{attribute 'no_explicit_call' := 'Do not call the body - Stick to OOP'}
FUNCTION_BLOCK FB_GigeCamera_Any EXTENDS FB_CH_Object IMPLEMENTS I_GevCameraControl, I_GigE_Beckhoff_Standalone, I_GetImage
VAR
	// This FB provides the basic functionality to control a GigE Vision camera and access its calibration data.
	fbCamera 						: FB_VN_GevCameraControl;	
	fbTriggerEtherCat				: FB_EtherCAT_Timestamp;
	
	{attribute 'hide'}	
	bInSimulation 					: BOOL;
	{attribute 'hide'}	
	eCameraType						: E_CameraType; 	
	{attribute 'hide'}
	fbGigeAnyRegister			 			: FB_GigE_Register_Any(ipCamera := THIS^);
	{attribute 'hide'}
	fbGigeBeckhoffRegisterVCS2xxx 			: FB_GigE_Register_Beckhoff_VCS2xxx(ipCamera := THIS^);
	{attribute 'hide'}
	fbGigeBeckhoffRegisterVUI2xxx 			: FB_GigE_Register_Beckhoff_VUI2xxx(ipCamera := THIS^);
	{attribute 'hide'}	
	ipRegister 								: I_GigeRegisterBase := fbGigeAnyRegister;
		
	{attribute 'hide'}	
	bInitDone 			: BOOL;
	{attribute 'hide'}
	bResetCommand		: BOOL;
	{attribute 'hide'}  						
	fbFeedback 			: FB_CH_Feedback(THIS^.fbSourceInfo); 
	{attribute 'hide'}
	fbAlarmOidNotSet 	: FB_TcAlarm;									// Alarm due to source state
	{attribute 'hide'}
	fbEthernetLinkDown 	: FB_TcAlarm;									// Camera is not connectode or has no power
	
	//TcCom object Camera
	{attribute 'hide'}
	ipGevImageProviderComObject 		: ITComObject;	
	{attribute 'hide'}
	ipGevImageAcquisitionComObject 		: ITComObject;	
	{attribute 'hide'}
	ipIpStackComObject 					: ITComObject;			
END_VAR

{attribute 'monitoring' := 'call'}
//Once as a Beckhoff camera is detected at startup, the corresponding type is loaded automatically. 
PROPERTY CameraType : E_CameraType
GET
CameraType := THIS^.eCameraType;
END_GET
SET
//if a new type is selectet, init the last one to reset all errors
IF (THIS^.CameraType <> THIS^.eCameraType) AND (THIS^.ipRegister <> 0) THEN
	THIS^.ipRegister.Initialize();
END_IF

//store new type
THIS^.eCameraType := CameraType;

//write new object to interface
CASE THIS^.eCameraType OF	
	E_CameraType.Beckhoff_VCS2xxx:
		THIS^.ipRegister := THIS^.fbGigeBeckhoffRegisterVCS2xxx;
		
	E_CameraType.Beckhoff_VUI2xxx:
		THIS^.ipRegister := THIS^.fbGigeBeckhoffRegisterVUI2xxx;
	
	ELSE
		THIS^.ipRegister := THIS^.fbGigeAnyRegister;;
END_CASE
END_SET
END_PROPERTY

//	The connection to the camera has been established. Gige-Vision parameters can now be read or written
{attribute 'monitoring' := 'call'}
PROPERTY ControlChannelOpen : BOOL
GET
CASE THIS^.State OF
	TCVN_CS_ERROR, TCVN_CS_INITIAL, TCVN_CS_INITIALIZING, TCVN_CS_INITIALIZED,TCVN_CS_OPENING,TCVN_CS_CLOSING:
		ControlChannelOpen := FALSE;
	
	TCVN_CS_OPENED, TCVN_CS_STARTACQUISITION,  TCVN_CS_ACQUIRING, TCVN_CS_STOPACQUISITION, TCVN_CS_RESETTINGFEATURES, TCVN_CS_TRIGGERING:
		ControlChannelOpen := TRUE;

	ELSE
		;//Unknown
END_CASE
END_GET
END_PROPERTY

METHOD FB_exit : BOOL
VAR_INPUT
	bInCopyCode : BOOL; // if TRUE, the exit method is called for exiting an instance that is copied afterwards (online change).
END_VAR
//Not on onlinechange
IF NOT bInCopyCode THEN
	IF THIS^.ipGevImageProviderComObject <> 0 THEN
		FW_SafeRelease(ADR(ipGevImageProviderComObject));
		FW_SafeRelease(ADR(ipGevImageAcquisitionComObject));
		FW_SafeRelease(ADR(ipIpStackComObject));
	END_IF	
END_IF
END_METHOD

METHOD FB_init : BOOL
VAR_INPUT
	bInitRetains : BOOL; // if TRUE, the retain variables are initialized (warm start / cold start)
	bInCopyCode : BOOL;  // if TRUE, the instance afterwards gets moved into the copy code (online change)
END_VAR
VAR
	fbGetCurTaskIdx  : GETCURTASKINDEX;
END_VAR
IF NOT bInCopyCode THEN
	//Start with an unknown camera. 
	//Once as a Beckhoff camera is detected, the corresponding type is loaded automatically. 
	THIS^.CameraType := E_CameraType.Unknown;
END_IF
END_METHOD

{attribute 'monitoring':='call'}
PROPERTY Feedback : I_CH_Feedback
GET
Feedback := THIS^.fbFeedback;
END_GET
END_PROPERTY

{attribute 'monitoring' := 'call'}
// This FB provides the basic functionality to control a GigE Vision camera and access its calibration data.
PROPERTY GevCameraControl : REFERENCE TO FB_VN_GevCameraControl
GET
GevCameraControl REF= THIS^.fbCamera;
END_GET
END_PROPERTY

METHOD Initialize : HRESULT
VAR 
	fbTaskInfo			: PlcTaskSystemInfo;
	nOid : OTCID;	
	nParaSize : UDINT;
	pParaData : PVOID;
	hr : HRESULT;
END_VAR
VAR_INST
	//This error cannot be reset. Requires a reset cold
	{attribute 'hide'}	
	fbInitError : FB_TcAlarm;
END_VAR
VAR CONSTANT
	N_IDX_OFFSET_GevImageAcquisition 	: UDINT := 16#00000001;
	N_IDX_OFFSET_IP_STACK 				: UDINT := 16#00000013;
END_VAR
hr := SUPER^.Initialize();


// Object id of ImagePoovider is not set
IF THIS^.fbCamera.oidITcVnGevImageProvider = 0 THEN
	IF NOT fbInitError.bRaised THEN 
		//This error cannot be reset. Requires a reset cold
		fbInitError.CreateEx(stEventEntry:=TC_EVENTS.CHALET_Vision_Events.ObjectIdNotSet, ipSourceInfo := THIS^.fbSourceInfo, bWithConfirmation := FALSE);
		fbInitError.Raise(0);
	END_IF
	Initialize := E_FAIL;
	RETURN;
END_IF


//Read information from TcCom object
//Get interface to ComObject
hr := FW_ObjMgr_GetObjectInstance(oid:= THIS^.OID, iid:= TC_GLOBAL_IID_LIST.IID_ITComObject, pipUnk:= ADR(THIS^.ipGevImageProviderComObject));
IF THIS^.ipGevImageProviderComObject <> 0 THEN
	//Read object id of TcCom GevImageAcquisitionComObject
	nOid := 0;
	nParaSize := SIZEOF(nOid);	pParaData := ADR(nOid);
	hr := ipGevImageProviderComObject.TcGetObjPara(pid:=N_IDX_OFFSET_GevImageAcquisition , nData:= nParaSize, pData:= pParaData, pgp:=0 );
	
	//Get interface of GevImageAcquisition
	hr := FW_ObjMgr_GetObjectInstance(oid:= nOid, iid:= TC_GLOBAL_IID_LIST.IID_ITComObject, pipUnk:= ADR(THIS^.ipGevImageAcquisitionComObject));
	IF THIS^.ipGevImageAcquisitionComObject <> 0 THEN
		//Read object id of TcCom 
		nOid := 0;
		nParaSize := SIZEOF(nOid);	pParaData := ADR(nOid);
		hr := ipGevImageAcquisitionComObject.TcGetObjPara(pid:=N_IDX_OFFSET_IP_STACK , nData:= nParaSize, pData:= pParaData, pgp:=0 );
		// If IP-Stack was not found in GevImageAcquisitionComObject then camera is in simulation mode
		IF hr = S_OK THEN
			//get interface to ipstack
			hr := FW_ObjMgr_GetObjectInstance(oid:= nOid, iid:= TC_GLOBAL_IID_LIST.IID_ITComObject, pipUnk:= ADR(THIS^.ipIpStackComObject));
		ELSE
			bInSimulation := TRUE;
			hr := S_OK;
		END_IF
	END_IF
END_IF


//Subelement
hr := GetMostSignificant(hr, fbTriggerEtherCat.Initialize());
IF THIS^.ipRegister <> 0 THEN
	hr := GetMostSignificant(hr, THIS^.ipRegister.Initialize());
END_IF


Initialize := hr;

IF Initialize = S_OK THEN
	THIS^.bInitDone := TRUE;
END_IF
END_METHOD

{attribute 'monitoring':='call'}
PROPERTY Initialized : BOOL
GET
Initialized := THIS^.bInitDone;
END_GET
END_PROPERTY

{attribute 'monitoring' := 'call'}
//Returns the OTCID OF the camera object.
PROPERTY OID : CHALET_BaseComponents.OTCID
GET
OID := THIS^.fbCamera.oidITcVnGevImageProvider;
END_GET
END_PROPERTY

{attribute 'monitoring' := 'call'}
// Module started successfully and entered aquiring mode
PROPERTY PUBLIC Operational : BOOL
GET
VAR
	eState : ETcVnCameraState;
END_VAR
eState := THIS^.State;
Operational := (eState = TCVN_CS_ACQUIRING) OR (eState = TCVN_CS_TRIGGERING);
END_GET
END_PROPERTY

{attribute 'monitoring' := 'call'}
//Access to the important parameters marked as standard in Gige-Vision
PROPERTY RegisterAnyCamera : I_GigE_Any_Camera
GET
//Convert in requestet interface
__QUERYINTERFACE(THIS^.ipRegister, RegisterAnyCamera);
END_GET
END_PROPERTY

{attribute 'monitoring' := 'call'}
//Interface to the parameters, can be 0(=invalid interface) depending on the hardware
PROPERTY RegisterBeckhoffCamera : I_GigE_Beckhoff_Camera
GET
//Convert in requestet interface
__QUERYINTERFACE(THIS^.ipRegister, RegisterBeckhoffCamera);
END_GET
END_PROPERTY

{attribute 'monitoring' := 'call'}
//Interface to the parameters, can be 0(=invalid interface) depending on the hardware
PROPERTY RegisterLighting : I_GigE_Beckhoff_Lighting
GET
//Convert in requestet interface
__QUERYINTERFACE(THIS^.ipRegister, RegisterLighting);
END_GET
END_PROPERTY

{attribute 'monitoring' := 'call'}
//Interface to the parameters, can be 0(=invalid interface) depending on the hardware
PROPERTY RegisterOpticControl : I_GigE_Beckhoff_OpticControl
GET
//Convert in requestet interface
__QUERYINTERFACE(THIS^.ipRegister, RegisterOpticControl);
END_GET
END_PROPERTY

//Try to reset the camera connection
METHOD Reset : HRESULT
VAR_INPUT
END_VAR
THIS^.bResetCommand := TRUE;

fbFeedback.ActiveCommand := 'Reset';
fbFeedback.LastCommandAccepted	:= TRUE;
fbFeedback.hr := THIS^.fbCamera.Reset();
END_METHOD

{attribute 'monitoring' := 'call'}
//Simulation mode is active
PROPERTY Simulation : BOOL
GET
Simulation := bInSimulation;
END_GET
END_PROPERTY

{attribute 'monitoring' := 'call'}
//Gets the current state of the internal camera control state machine.
PROPERTY State : ETcVnCameraState
GET
State := THIS^.fbCamera.GetState();
END_GET
END_PROPERTY

{attribute 'monitoring' := 'call'}
//Access to the interface to control the EtherCAT timestamp trigger
PROPERTY TriggerEtherCat : I_EtherCat_Trigger
GET
TriggerEtherCat := THIS^.fbTriggerEtherCat;
END_GET
END_PROPERTY

//Send the 'SoftwareTriggerCommands' defined in the TcVnGevImageProvider TcCOM module to the camera.
METHOD PUBLIC TriggerSoftware : HRESULT
VAR
	eState : ETcVnCameraState;
END_VAR
eState := THIS^.State;

(* Check if not in wrong state *)
IF NOT ((eState = ETcVnCameraState.TCVN_CS_ACQUIRING) OR (eState = ETcVnCameraState.TCVN_CS_OPENED) OR THIS^.Simulation) THEN
	TriggerSoftware := E_FAIL;
	RETURN;
END_IF

// Trigger image
fbFeedback.ActiveCommand := 'TriggerImage';
fbFeedback.LastCommandAccepted	:= TRUE;
fbFeedback.hr := fbCamera.TriggerImage();
TriggerSoftware := fbFeedback.hr;
END_METHOD

//Gets the current available image (first in receive queue) and its corresponding GVSP info
METHOD TryGetImage : HRESULT
VAR_INPUT
	stImageWithInfo : REFERENCE TO ST_ImageWithInfo;
END_VAR
VAR_INST
	{attribute 'hide'}							
    fbCrititcalSection : FB_IecCriticalSection;    						// Internal lock for test & set function    
END_VAR
VAR
	ipImageTemp   : ITcVnImage;
	stGvspInfoTemp : GVSP_IMAGE_INFO;
END_VAR
IF NOT __ISVALIDREF(stImageWithInfo) THEN
	//Error, invalide input
	TryGetImage := E_FAIL;
	RETURN;
END_IF


(*  Lock the image to prevent multiple access *)
(*	🔒 LOCKED FROM HERE --------------------------------------------- *)
IF fbCrititcalSection.Enter() THEN
	
	(* Get current image from camera and store result in temp variable*)
	TryGetImage := fbCamera.GetCurrentImageWithGvspInfo(
						ipImage := ipImageTemp,
						stGvspInfo := stGvspInfoTemp
						);
					
	(* If new image found *)				
	IF TryGetImage = S_OK THEN
		
		(* Release the old image before overwriting it with the new one *)	
		IF stImageWithInfo.ipImage <> 0 THEN
			FW_SafeRelease(ADR(stImageWithInfo.ipImage));
		END_IF		
	
		//Handover new data
		stImageWithInfo.ipImage 		:= ipImageTemp;
		stImageWithInfo.stGvspInfo 		:= stGvspInfoTemp;

		(*For a camera a fictitious name *)
		stImageWithInfo.sCurrentImageFileName := TO_STRING(stImageWithInfo.stGvspInfo.BlockId);		

		
		(* Get image info from received image *)
		F_VN_GetImageInfo(	ipImage:=stImageWithInfo.ipImage, 
							stImageInfo:=stImageWithInfo.stInfo, 
							hrPrev:=TryGetImage );	
	END_IF



	(*	🔓 LOCKED TO HERE ----------------------------------------------- *)
	fbCrititcalSection.Leave();
END_IF
END_METHOD

METHOD Update : HRESULT
VAR
	ipVnRegisterStatus : I_VnRegister;
	bAllReadDone : BOOL := TRUE;
	bAllWriteDone : BOOL := TRUE;
	nParaSize : UDINT;
	pParaData : PVOID;
	hr : HRESULT;
	stIpStackData : ST_IpStackDiag;
	bLinkDetected : BOOL;
	bParaReadSuccessful : BOOL;
END_VAR
VAR CONSTANT
	N_IDX_OFFSET_IP_STACK 	: UDINT := 16#03011108; // Parameter(online) in Planar Track object
END_VAR
//Force to initialize first
IF NOT THIS^.Initialized THEN
	THIS^.Initialize();
	RETURN;
END_IF


(* Source state machine *)
CASE THIS^.State OF
	TCVN_CS_INITIAL, TCVN_CS_INITIALIZING:
		fbFeedback.ActiveCommand := 'InitializeCamera';
		fbFeedback.hr := fbCamera.InitializeCamera();

	TCVN_CS_INITIALIZED,  TCVN_CS_OPENING:	
		IF THIS^.ipRegister <> 0 THEN
			//Redo a read or write for each parameter
			THIS^.ipRegister.RewriteParameters();
		END_IF
		fbFeedback.ActiveCommand := 'OpenCamera';
		fbFeedback.hr := fbCamera.OpenCamera();
		
	TCVN_CS_OPENED:
		(* Detect camera model once if unknown *)
		IF THIS^.CameraType = E_CameraType.Unknown AND THIS^.RegisterAnyCamera <> 0 AND THIS^.ipRegister.AllReadDone THEN
			IF FIND(THIS^.RegisterAnyCamera.DeviceModeNamel, 'VCS2') <> 0 THEN
				THIS^.CameraType := E_CameraType.Beckhoff_VCS2xxx;
			ELSIF FIND(THIS^.RegisterAnyCamera.DeviceModeNamel, 'VUI2') <> 0 THEN
				THIS^.CameraType := E_CameraType.Beckhoff_VUI2xxx;
			ELSE
				THIS^.CameraType := E_CameraType.ThirdParty;
			END_IF
		END_IF
		
		IF THIS^.Simulation THEN
			; //Stay in this state in Simulationmode	
		
		ELSIF THIS^.ipRegister = 0 THEN
			fbFeedback.ActiveCommand := 'StartAcquisition';
			fbFeedback.hr := fbCamera.StartAcquisition();
			
		ELSIF THIS^.ipRegister.AllReadDone AND THIS^.ipRegister.AllWriteDone THEN
			fbFeedback.ActiveCommand := 'StartAcquisition';
			fbFeedback.hr := fbCamera.StartAcquisition();

		ELSE	
			//Read and write all camera parameter in this OPENED-State 
			fbFeedback.ActiveCommand := 'ReadWrite camera parameters';
			fbFeedback.Busy	:= TRUE;
		END_IF
	
		
	TCVN_CS_STARTACQUISITION:
		fbFeedback.ActiveCommand := 'StartAcquisition';
		fbFeedback.hr := fbCamera.StartAcquisition();
		
		
	TCVN_CS_STOPACQUISITION:
		fbFeedback.ActiveCommand := 'StopAcquisition';
		fbFeedback.hr := fbCamera.StopAcquisition();
		
	TCVN_CS_ACQUIRING:
		;//wait for trigger
		
		//Check if a chage in opened state is required to read/write parameter
		IF VisionParameterlist.B_LEAVE_AQUIRRING_STATE_TO_WRITE_PARAMETER AND THIS^.ipRegister <> 0 AND_THEN NOT THIS^.ipRegister.AllWriteDone THEN
			fbFeedback.ActiveCommand := 'StopAcquisition';
			fbCamera.StopAcquisition();
		END_IF
		
	TCVN_CS_TRIGGERING:
		(* Execute the triggering until done *)
		fbFeedback.ActiveCommand := 'TriggerImage';
		fbFeedback.hr := fbCamera.TriggerImage();
		
	TCVN_CS_ERROR:	
		(* Reset if commanded *)
		IF THIS^.bResetCommand THEN
			fbFeedback.ActiveCommand := 'Reset';
			fbFeedback.hr := THIS^.fbCamera.Reset();			
		END_IF
		
END_CASE

(* Clear reset request if not in Error-State *)
IF THIS^.State <> TCVN_CS_ERROR THEN
	THIS^.bResetCommand := FALSE;
END_IF




// --- Write diagnostic information to eventloger
IF THIS^.State = TCVN_CS_ERROR AND VisionParameterlist.B_ALARM_IF_LINK_TO_CAMERA_IS_DOWN THEN
	//check IP-Stack an check if camera is conected	
	IF THIS^.ipIpStackComObject <> 0 THEN
		//Read object id of ipStack TcCom 
		nParaSize := SIZEOF(stIpStackData);	pParaData := ADR(stIpStackData);
		hr := ipIpStackComObject.TcGetObjPara(	pid		:=N_IDX_OFFSET_IP_STACK , 
												nData	:= nParaSize, 
												pData	:= pParaData, 
												pgp		:=0 );
		
		 // Link is active on uneven cts of linkchanges
		bLinkDetected := (stIpStackData.nLinkStatusChangedCnt MOD 2) = 1;
		bParaReadSuccessful := hr = S_OK;
		IF NOT THIS^.Simulation AND bParaReadSuccessful AND NOT bLinkDetected AND NOT fbEthernetLinkDown.bRaised THEN
			fbEthernetLinkDown.CreateEx(stEventEntry 		:= TC_EVENTS.CHALET_Vision_Events.EthernetLinkDown,
										ipSourceInfo 		:= THIS^.fbSourceInfo,
										bWithConfirmation 	:= FALSE);
			fbEthernetLinkDown.Raise(0);			
	
		ELSIF fbEthernetLinkDown.bRaised AND (THIS^.Simulation AND NOT bParaReadSuccessful OR bLinkDetected) THEN
			fbEthernetLinkDown.Clear(0,0);		
			
		ELSE
			; //nothing
		END_IF
	END_IF
END_IF


//Subelement - if not in simulation
fbTriggerEtherCat.Update();

IF THIS^.ipRegister <> 0 THEN
	//Redo a read or write for each parameter
	THIS^.ipRegister.Update();
END_IF
END_METHOD

END_FUNCTION_BLOCK

(* stored: Version 1.1.0.1, ProductVersion 3.1.4026.19
   POU FB_GigeCamera_Any: Id {e8c292d8-c8f1-47c5-8349-a7443f582da7}, SpecialFunc None
   Property CameraType: Id {7fb62898-c1ef-473f-8fa5-37fc744dfaeb}
   Get Get: Id {6fbdc49f-5dec-49b6-b3b2-6ecf421f6204}
   Set Set: Id {f1d50843-b071-4042-b7c8-71452311f410}
   Property ControlChannelOpen: Id {9ac1a404-f3db-4ca1-8cf3-21dcc8494d47}
   Get Get: Id {18acef6b-5a92-4cac-8fe9-f38fe5906b7c}
   Method FB_exit: Id {22a0fd36-0f2b-40fc-a0b7-e0a470e76283}
   Method FB_init: Id {6d48896f-0163-44cc-930b-b0132ca2b6f1}
   Property Feedback: Id {25a83ed1-35db-403a-8b79-b1707e7b3bf5}
   Get Get: Id {05de5582-afd6-49ee-8b6a-a404cc9a5153}
   Property GevCameraControl: Id {a6a5ff40-e698-4eb9-a4af-7e7b956de53b}
   Get Get: Id {4dbcaeb3-d198-410e-97c9-10d4ba383e48}
   Method Initialize: Id {bc3ff501-3767-4510-b98a-2583f7f1bf51}
   Property Initialized: Id {178783fa-217d-4798-9b8e-d70049fcf541}
   Get Get: Id {56ce6899-32d2-404f-b92a-ec207c58a345}
   Property OID: Id {d45d7cb9-9db9-405f-b0dc-b7829281ff91}
   Get Get: Id {56913cf9-4381-4276-9512-01359e1a5425}
   Property Operational: Id {9b1561a2-3115-4016-a31a-87faf9e28f65}
   Get Get: Id {6d77fdf6-f25e-4c00-846a-cd2fdd7d4509}
   Property RegisterAnyCamera: Id {8d567bcb-298b-442f-a2ee-91a6c021730c}
   Get Get: Id {0420c097-062d-482b-8cb1-5ce6c81ddc73}
   Property RegisterBeckhoffCamera: Id {7006d77f-1177-4d8f-8d2e-4799aa5ef962}
   Get Get: Id {56e40d86-31f2-4a86-b952-e35c1b162e6c}
   Property RegisterLighting: Id {3bc93099-1af4-4df9-a214-2075b055cd4e}
   Get Get: Id {85ef6c0e-3835-4f12-b3d4-c1e462184f60}
   Property RegisterOpticControl: Id {480374a2-f3ac-43eb-951f-9329e1d1b209}
   Get Get: Id {4c574dc9-5086-42a5-9522-7829f29520e1}
   Method Reset: Id {3060e3a3-a4a0-40c3-95ce-133e9b21bdc7}
   Property Simulation: Id {f5897538-8906-4a6c-a04c-f5219ee092c3}
   Get Get: Id {e545d061-2cf2-4952-931a-feba73b0f494}
   Property State: Id {50e80ae9-2935-4fb3-9258-b3bc964b950f}
   Get Get: Id {403fa147-7caa-45cc-b95d-19e7e59994e7}
   Property TriggerEtherCat: Id {d56cc878-4ab2-4eaf-906d-a4f6451fdf4c}
   Get Get: Id {5511c542-b995-4328-b8d3-a625ef59ee40}
   Method TriggerSoftware: Id {eebc06d9-4bb8-48c3-8885-1edcdf59cd74}
   Method TryGetImage: Id {a7872ab3-e0b7-44ca-a9ad-ab28324c5ff8}
   Method Update: Id {f47126a0-8dd0-475c-9002-45ef62606169} *)
